{attribute 'qualified_only'}
//{attribute 'strict'}
TYPE ConveyorMode :
(
	IDLE,
	FORWARD,
	BACKWARD,
	STOP,
	
	size
);
END_TYPE

(* stored: Version 1.1.0.1, ProductVersion 3.1.4024.11
   DUT ConveyorMode: Id {ae925df4-5321-4234-bd5c-a6ddfde7cc36} *)
